// TIA Portal project "Control de subida y bajada de una cortina con HMI" (V15.1)

(* hardware
DEVICE "S7-1200 station_1"  S7-1200 Station
   slot 0: "Rack_0"  S7-1200 Rack  Rack  V1.0
   slot 1: "PLC_1"  CPU 1212C AC/DC/Rly  6ES7 212-1BD30-0XB0  V2.2
      slot 3: "AQ 1x12BIT_1"  AQ1 signal board  6ES7 232-4HA30-0XB0  V1.0
DEVICE "HMI_1"  KTP400 Basic PN
   slot 0: "KTP400 Basic PN"  KTP400 Basic PN  6AV2 123-2DB03-0AX0  14.0.0.0
   slot 1: "HMI_RT_1"  KTP400 Basic PN  6AV2 123-2DB03-0AX0  14.0.0.0
   slot 5: "HMI_1.IE_CP_1"  PROFINET Interface  14.0.0.0
      slot 1: "Interfaz PROFINET_1"  PROFINET Interface
         slot 1: "Port_1"  Port
*)

// ===== PLC "PLC_1"  CPU 1212C AC/DC/Rly =====

VAR_GLOBAL   // PLC tag table "Tabla de variables estándar"
   "Abrir cortina" AT %M0.0 : Bool;
   "Cerrar cortina" AT %M0.1 : Bool;
   "Arrancar motor" AT %Q0.0 : Bool;
   "Sentido del motor" AT %Q0.1 : Bool;
   "Sensor high" AT %I0.0 : Bool;
   "Sensor low" AT %I0.1 : Bool;
   "Entrada analogica 0" AT %IW64 : Int;
   "dato" AT %MW2 : Int;
END_VAR

ORGANIZATION_BLOCK "Main"   // OB1, LAD, ProgramCycle
TITLE = "Main Program Sweep (Cycle)"
{ S7_Optimized_Access := 'TRUE' }
VERSION : 0.1
   VAR_TEMP
      Activarcortina1 : Bool;
      Cerrarcortina1 : Bool;
   END_VAR
BEGIN

REGION Network 1
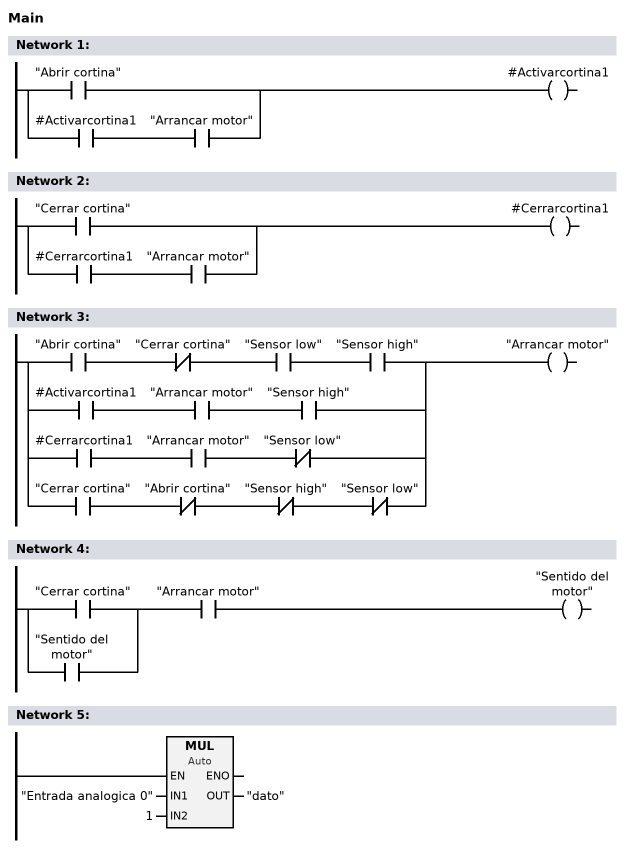
   RUNG wire#powerrail
      Contact( "Abrir cortina" )
      wire#w1
      Coil( #Activarcortina1 )
   END_RUNG
   RUNG wire#powerrail
      Contact( #Activarcortina1 )
      Contact( "Arrancar motor" )
   END_RUNG wire#w1
   // the same network as SCL:
   #Activarcortina1 := "Abrir cortina" OR (#Activarcortina1 AND "Arrancar motor");
END_REGION

REGION Network 2
   RUNG wire#powerrail
      Contact( "Cerrar cortina" )
      wire#w1
      Coil( #Cerrarcortina1 )
   END_RUNG
   RUNG wire#powerrail
      Contact( #Cerrarcortina1 )
      Contact( "Arrancar motor" )
   END_RUNG wire#w1
   // the same network as SCL:
   #Cerrarcortina1 := "Cerrar cortina" OR (#Cerrarcortina1 AND "Arrancar motor");
END_REGION

REGION Network 3
   RUNG wire#powerrail
      Contact( "Abrir cortina" )
      I_Contact( "Cerrar cortina" )
      Contact( "Sensor low" )
      Contact( "Sensor high" )
      wire#w1
      Coil( "Arrancar motor" )
   END_RUNG
   RUNG wire#powerrail
      Contact( #Activarcortina1 )
      Contact( "Arrancar motor" )
      Contact( "Sensor high" )
   END_RUNG wire#w1
   RUNG wire#powerrail
      Contact( #Cerrarcortina1 )
      Contact( "Arrancar motor" )
      I_Contact( "Sensor low" )
   END_RUNG wire#w1
   RUNG wire#powerrail
      Contact( "Cerrar cortina" )
      I_Contact( "Abrir cortina" )
      I_Contact( "Sensor high" )
      I_Contact( "Sensor low" )
   END_RUNG wire#w1
   // the same network as SCL:
   "Arrancar motor" := ("Abrir cortina" AND NOT "Cerrar cortina" AND "Sensor low" AND "Sensor high") OR (#Activarcortina1 AND "Arrancar motor" AND "Sensor high") OR (#Cerrarcortina1 AND "Arrancar motor" AND NOT "Sensor low") OR ("Cerrar cortina" AND NOT "Abrir cortina" AND NOT "Sensor high" AND NOT "Sensor low");
END_REGION

REGION Network 4
   RUNG wire#powerrail
      Contact( "Cerrar cortina" )
      wire#w1
      Contact( "Arrancar motor" )
      Coil( "Sentido del motor" )
   END_RUNG
   RUNG wire#powerrail
      Contact( "Sentido del motor" )
   END_RUNG wire#w1
   // the same network as SCL:
   "Sentido del motor" := ("Cerrar cortina" OR "Sentido del motor") AND "Arrancar motor";
END_REGION

REGION Network 5
   RUNG wire#powerrail
      { S7_GenerateENO := "TRUE" } Mul(in1 := "Entrada analogica 0", in2 := 1, out => "dato")
   END_RUNG
   // the same network as SCL:
   "dato" := "Entrada analogica 0" * 1;
END_REGION
END_ORGANIZATION_BLOCK

(* ===== HMI "HMI_RT_1" =====
system functions are stored by id; their names below are inferred from use
connection "HMI_Conexión_1": ETHERNET, SMART_S7_1200_OMS

HMI tags "Tabla de variables estándar"
   "Número_imagen_variable" : UInt, internal
   "Abrir cortina" : Bool = PLC "Abrir cortina" AT %M0.0, 1 s
   "Cerrar cortina" : Bool = PLC "Cerrar cortina" AT %M0.1, 1 s
   "Sensor high" : Bool = PLC "Sensor high" AT %I0.0, 1 s
   "Sensor low" : Bool = PLC "Sensor low" AT %I0.1, 1 s

text list "Nombre_imagen_lista_texto": 1 'Imagen raíz'

Template "Plantilla_1" 480x272
   Button "Template_Button" at 415,46 size 63x44; TextOff 'Text'
   Button "Template_Button_1" at 415,91 size 63x44; TextOff 'Text'
   Button "Template_Button_2" at 415,136 size 63x44; TextOff 'Text'
   Button "Template_Button_3" at 415,181 size 63x44; TextOff 'Text'
   Button "Template_Button_4" at 415,226 size 63x44; TextOff 'Text'
   SymbolicIOField "Imagen_campo_ES_simbólico" at 2,8 size 391x29; TextOff '0'; TextOn '1'; TextList "Nombre_imagen_lista_texto"
      ProcessValue <- "Número_imagen_variable"
      on Change: ActivateScreenByNumber("Número_imagen_variable", 0)
   DateTimeField "HmiScreenItemData" at 395,22 size 85x22
   DateTimeField "HmiScreenItemData_1" at 395,0 size 85x22

screen "Imagen raíz" 480x272, template "Plantilla_1"
   on GenerateScreen: SetTag("Número_imagen_variable", 1)
   Button "Botón_1" at 58,85 size 96x32; TextOff 'Abrir cortina'
      on Press: function_b14e0dd5("Abrir cortina", 0)
   Button "Botón_2" at 286,85 size 96x32; TextOff 'Cerrar cortina'
      on Press: function_b14e0dd5("Cerrar cortina", 0)
   Circle "Círculo_1" at 197,117 size 48x48
      Visibility <- "Sensor high"
   Circle "Círculo_2" at 197,181 size 48x48
      Visibility <- "Sensor low"
   TextField "Campo de texto_1" at 250,130 size 79x20; Text 'Sensor alto'
   TextField "Campo de texto_2" at 250,196 size 82x20; Text 'Sensor bajo'
*)